FUNCTION_BLOCK ExampleDomain_States
VAR_OUTPUT
	iExample		: I_Tag;
END_VAR

END_FUNCTION_BLOCK

(* stored: Version 1.1.0.1
   POU ExampleDomain_States: Id {e8ee2b6b-9190-4317-9c0f-e43666986367}, SpecialFunc None *)
